// TIA Portal project "Plantilla_PID-FactoryIO" (V14)

(* hardware
DEVICE "S71500/ET200MP-Station_1"  S7-1500 station
   slot 0: "Profilschiene_0"  6ES7 590-1***0-0AA0
   slot 1: "PLC_1"  CPU 1511-1 PN  6ES7 511-1AK00-0AB0  V1.8
   slot 2: "AI 8xU/I/RTD/TC ST_1"  AI 8xU/I/RTD/TC ST  6ES7 531-7KF00-0AB0  V2.0
   slot 3: "AI 8xU/I/RTD/TC ST_2"  AI 8xU/I/RTD/TC ST  6ES7 531-7KF00-0AB0  V2.0
   slot 4: "AI 8xU/I/RTD/TC ST_3"  AI 8xU/I/RTD/TC ST  6ES7 531-7KF00-0AB0  V2.0
   slot 5: "AI 8xU/I/RTD/TC ST_4"  AI 8xU/I/RTD/TC ST  6ES7 531-7KF00-0AB0  V2.0
   slot 6: "DI 16x24VDC BA_1"  DI 16x24VDC BA  6ES7 521-1BH10-0AA0  V1.0
*)

// ===== PLC "PLC_1"  CPU 1511-1 PN =====

VAR_GLOBAL   // PLC tag table "IO"
   "Arranque" AT %I0.0 : Bool;
   "Reset" AT %I0.1 : Bool;
   "Parada" AT %I0.2 : Bool;
   "Luz Arranque" AT %Q0.0 : Bool;
   "Luz Reset" AT %Q0.1 : Bool;
   "Luz Parada" AT %Q0.2 : Bool;
   "Sensor de nivel" AT %ID30 : Real;
   "Caudalímetro" AT %ID34 : Real;
   "Consigna" AT %ID38 : Real;
   "Válvula de llenado" AT %QD30 : Real;
   "Válvula de vaciado" AT %QD34 : Real;
   "Indicador Consigna" AT %QD38 : DInt;
   "Indicador Nivel" AT %QD42 : DInt;
   "Habilitacion PID" AT %M0.0 : Bool;
   "SP Manual" AT %ID42 : Real;
   "Indicador SP Manual" AT %QD46 : DInt;
END_VAR

FUNCTION "MHJ-PLC-Lab-Function-S71500" : Void   // FC9000, SCL
{ S7_Optimized_Access := 'TRUE' }
VERSION : 0.1
   VAR_TEMP
      Value : Byte;
      ForCounter : Int;
   END_VAR
   VAR CONSTANT
      Value_01_DW : DWord := 16#1223_5486;
      Value_02_DW : DWord := 16#A6C9_D1F5;
   END_VAR
BEGIN

   #Value:=PEEK(area := 16#82,
        dbNumber := 0,
        byteOffset := 511);
   #Value := #Value + 1;

   POKE(area := 16#82,
        dbNumber := 0,
        byteOffset := 511,
        value := #Value);

   POKE(area := 16#82,
        dbNumber := 0,
        byteOffset := 1016,
        value := #Value_01_DW);
   POKE(area := 16#82,
        dbNumber := 0,
        byteOffset := 1020,
        value := #Value_02_DW);

   FOR #ForCounter := 0 TO 63 DO
       #Value:=PEEK(area := 16#1,
            dbNumber := 0,
            byteOffset := #ForCounter);
       POKE(area := 16#81,
            dbNumber := 0,
            byteOffset := #ForCounter,
            value := #Value);
   END_FOR;
   #Value := PEEK(area := 16#1,
                  dbNumber := 0,
                  byteOffset := 512);
   POKE(area := 16#82,
        dbNumber := 0,
        byteOffset := 512,
        value := #Value);
END_FUNCTION

ORGANIZATION_BLOCK "Main"   // OB1, FBD, ProgramCycle
TITLE = "Main Program Sweep (Cycle)"
{ S7_Optimized_Access := 'TRUE' }
VERSION : 0.1
   VAR_INPUT
      Initial_Call : Bool;   // Initial call of this OB
      Remanence : Bool;   // =True, if remanent data are available
   END_VAR
BEGIN

REGION Network 1
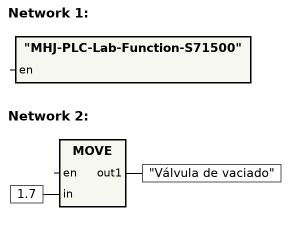
   "MHJ-PLC-Lab-Function-S71500"();
END_REGION

REGION Network 2
   "Válvula de vaciado" := 1.7;
END_REGION
END_ORGANIZATION_BLOCK

ORGANIZATION_BLOCK "Cyclic interrupt"   // OB30, LAD, CyclicInterrupt
{ S7_Optimized_Access := 'TRUE' }
VERSION : 0.1
   VAR_INPUT
      Initial_Call : Bool;   // Initial call of this OB
      Event_Count : Int;   // Events discarded
   END_VAR
   VAR_TEMP
      Nivel_ESC : Real;
      Consigna_ESC : Real;
      SP_MAN_ESC : Real;
      Valvula_REAL : Real;
   END_VAR
BEGIN

REGION Network 1: Escalados
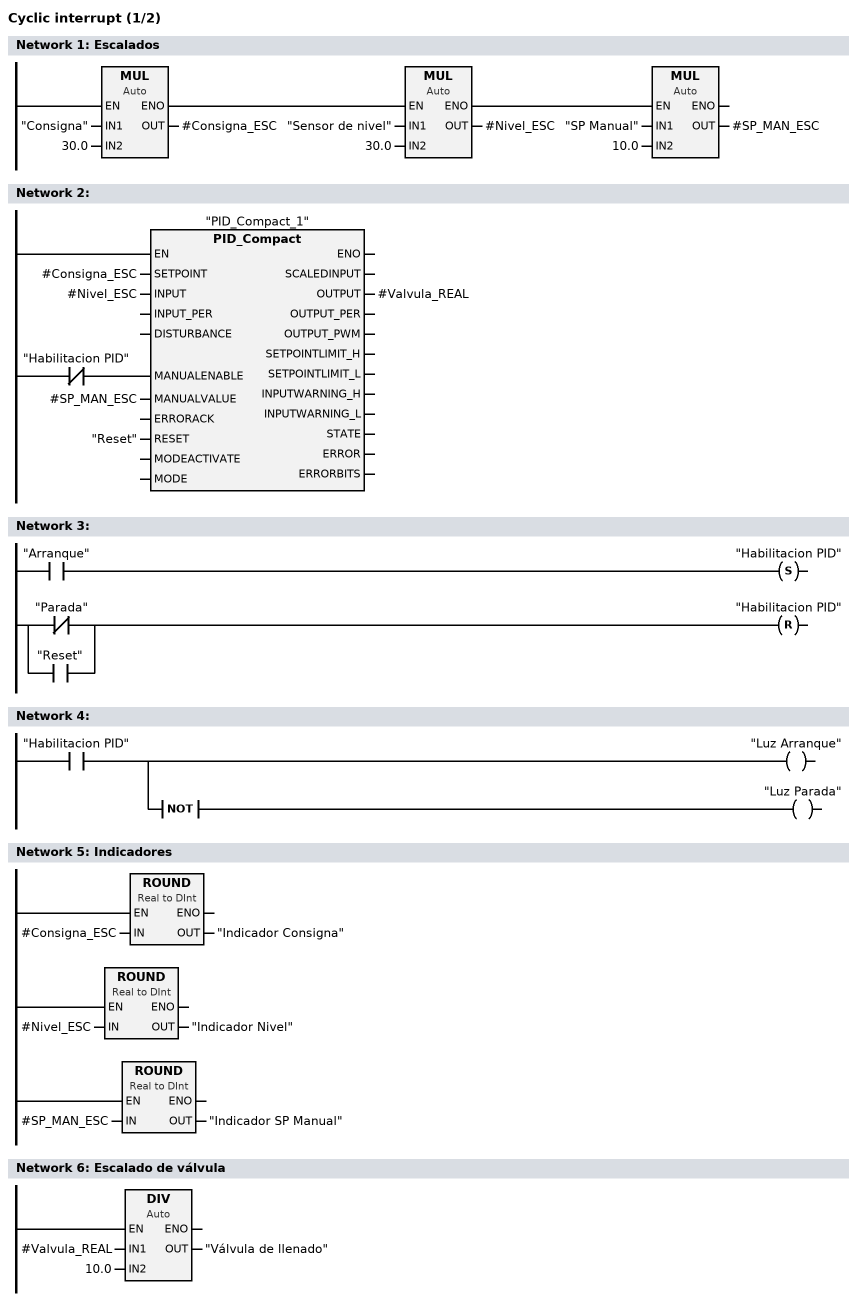
   RUNG wire#powerrail
      Mul(in1 := "Consigna", in2 := 30.0, out => #Consigna_ESC)
      Mul(in1 := "Sensor de nivel", in2 := 30.0, out => #Nivel_ESC)
      Mul(in1 := "SP Manual", in2 := 10.0, out => #SP_MAN_ESC)
   END_RUNG
   // the same network as SCL:
   #Consigna_ESC := "Consigna" * 30.0;
   #Nivel_ESC := "Sensor de nivel" * 30.0;
   #SP_MAN_ESC := "SP Manual" * 10.0;
END_REGION

REGION Network 2
   "PID_Compact_1"(Setpoint := #Consigna_ESC,   // PID_Compact
                   Input := #Nivel_ESC,
                   ManualEnable := NOT "Habilitacion PID",
                   ManualValue := #SP_MAN_ESC,
                   Reset := "Reset",
                   Output => #Valvula_REAL);
END_REGION

REGION Network 3
   RUNG wire#powerrail
      Contact( "Arranque" )
      S_Coil( "Habilitacion PID" )
   END_RUNG
   RUNG wire#powerrail
      I_Contact( "Parada" )
      wire#w1
      R_Coil( "Habilitacion PID" )
   END_RUNG
   RUNG wire#powerrail
      Contact( "Reset" )
   END_RUNG wire#w1
   // the same network as SCL:
   IF "Arranque" THEN "Habilitacion PID" := TRUE; END_IF;
   IF NOT "Parada" OR "Reset" THEN "Habilitacion PID" := FALSE; END_IF;
END_REGION

REGION Network 4
   RUNG wire#powerrail
      Contact( "Habilitacion PID" )
      wire#w1
      Coil( "Luz Arranque" )
   END_RUNG
   RUNG wire#w1
      Not()
      Coil( "Luz Parada" )
   END_RUNG
   // the same network as SCL:
   "Luz Arranque" := "Habilitacion PID";
   "Luz Parada" := NOT "Habilitacion PID";
END_REGION

REGION Network 5: Indicadores
   RUNG wire#powerrail
      { S7_Templates := "[SrcType := Real, DestType := DInt]" } Round(in := #Consigna_ESC, out => "Indicador Consigna")
   END_RUNG
   RUNG wire#powerrail
      { S7_Templates := "[SrcType := Real, DestType := DInt]" } Round(in := #Nivel_ESC, out => "Indicador Nivel")
   END_RUNG
   RUNG wire#powerrail
      { S7_Templates := "[SrcType := Real, DestType := DInt]" } Round(in := #SP_MAN_ESC, out => "Indicador SP Manual")
   END_RUNG
   // the same network as SCL:
   "Indicador Consigna" := ROUND(#Consigna_ESC);
   "Indicador Nivel" := ROUND(#Nivel_ESC);
   "Indicador SP Manual" := ROUND(#SP_MAN_ESC);
END_REGION

REGION Network 6: Escalado de válvula
   RUNG wire#powerrail
      Div(in1 := #Valvula_REAL, in2 := 10.0, out => "Válvula de llenado")
   END_RUNG
   // the same network as SCL:
   "Válvula de llenado" := #Valvula_REAL / 10.0;
END_REGION

REGION Network 7: enable monitoring of call cycle time
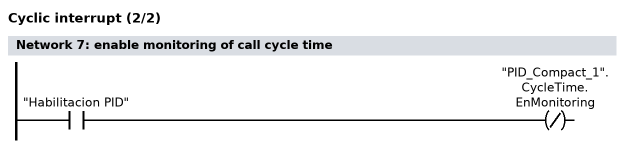
   RUNG wire#powerrail
      Contact( "Habilitacion PID" )
      I_Coil( "PID_Compact_1".CycleTime.EnMonitoring )
   END_RUNG
   // the same network as SCL:
   "PID_Compact_1".CycleTime.EnMonitoring := NOT "Habilitacion PID";
END_REGION
END_ORGANIZATION_BLOCK